PROGRAM P_Demo_FB_MBUdpWriteRegs
VAR
    fbUdpWriteRegs: FB_MBUdpWriteRegs;
    sTargetIp     : STRING(15) := '192.168.1.50';   // 目标 Modbus 设备 IP（按现场改）
    bTrigger      : BOOL;          // 在线置一次上升沿触发本次访问
    bBusy         : BOOL;          // 在线 monitor：执行中为 TRUE
    bError        : BOOL;          // 出错置 TRUE
    nErrId        : UDINT;         // 出错时的 ADS/Modbus 错误码
    arrData       : ARRAY [0..2] OF WORD := [100,200,300];   // 待写出的数据
END_VAR

// ============================================================
// Tc2_ModbusSrv.FB_MBUdpWriteRegs 演示程序（Modbus TCP 客户端 / 主站）
// ============================================================
// 场景：向设备一次性下发一组参数，例如给运动控制器写入一段轨迹点、给配方设备下发一组工艺参数（多个 16 位寄存器）。 选用 UDP 版多见于同一控制柜/同网段、对实时性敏感且能容忍偶发丢包的场景，省去 TCP 建链开销。
// 价值：批量写寄存器用功能码 16，一次报文写多个字；本 FB 把 `WORD` 数组一次写出，省去多次往返。
// 验证：登录后在线置 bTrigger := TRUE 触发一次；观察 bBusy 在数个周期后回 FALSE，
//       bError 应为 FALSE、nErrId 应为 0；若对端不在线则 bError=TRUE 且 nErrId 含超时码。
//       本例：一次写 3 个寄存器（一组工艺参数）
// 验证步骤：
//   1. 右键 PLC 项目下 POUs 文件夹 → Add → Existing Item → 选本 .TcPOU 文件
//   2. 引用 Tc2_ModbusSrv（References → Add library），并确保 TF6250 Modbus TCP 已授权运行
//   3. 把 sTargetIp 改成现场 Modbus 设备 IP；编译 → 登录 → 运行
//   4. 在线脉冲 bTrigger，按上方『验证』观察输出
// ============================================================

// 单次完整调用：所有 VAR_INPUT 显式赋值；bExecute 边沿触发一次
fbUdpWriteRegs(
    sIPAddr   := sTargetIp,
    nTCPPort  := MODBUS_TCP_PORT,
    nUnitID   := 16#FF,
    nQuantity := 3,
    nMBAddr   := 0,
    cbLength  := SIZEOF(arrData),
    pSrcAddr  := ADR(arrData),
    bExecute  := bTrigger,
    tTimeout  := T#5S,
    bBUSY     => bBusy,
    bError    => bError,
    nErrId    => nErrId
);

END_PROGRAM

(* stored: Version 1.1.0.1, ProductVersion 3.1.4024.5
   POU P_Demo_FB_MBUdpWriteRegs: Id {3d3c535d-94cc-5f29-be70-2d97cc4c1ba0}, SpecialFunc None *)
